{attribute addProperty BoxType "EJ2918-0000-0017"}
{attribute addProperty Id "Module_1_Channel_1_Standard_OutputAT %Q*BOOL811Module_1_Channel_2_Standard_OutputAT %Q*BOOL812Module_1_Channel_3_Standard_OutputAT %Q*BOOL813Module_1_Channel_4_Standard_OutputAT %Q*BOOL814Module_2_Channel_1_Standard_OutputAT %Q*BOOL811Module_2_Channel_2_Standard_OutputAT %Q*BOOL812Module_2_Channel_3_Standard_OutputAT %Q*BOOL813Module_2_Channel_4_Standard_OutputAT %Q*BOOL814"}
{attribute addProperty CRC "3397865097"}
{attribute addProperty SizeInBites "64"}
{attribute addProperty SizeInBytes "8"}
TYPE Outputs_CA874E89 :
STRUCT
	{attribute addProperty Name "Module_1_Channel_1_Standard_Output"}
	Module_1_Channel_1_Standard_Output AT %Q* : BOOL;
	{attribute addProperty Name "Module_1_Channel_2_Standard_Output"}
	Module_1_Channel_2_Standard_Output AT %Q* : BOOL;
	{attribute addProperty Name "Module_1_Channel_3_Standard_Output"}
	Module_1_Channel_3_Standard_Output AT %Q* : BOOL;
	{attribute addProperty Name "Module_1_Channel_4_Standard_Output"}
	Module_1_Channel_4_Standard_Output AT %Q* : BOOL;
	{attribute addProperty Name "Module_2_Channel_1_Standard_Output"}
	Module_2_Channel_1_Standard_Output AT %Q* : BOOL;
	{attribute addProperty Name "Module_2_Channel_2_Standard_Output"}
	Module_2_Channel_2_Standard_Output AT %Q* : BOOL;
	{attribute addProperty Name "Module_2_Channel_3_Standard_Output"}
	Module_2_Channel_3_Standard_Output AT %Q* : BOOL;
	{attribute addProperty Name "Module_2_Channel_4_Standard_Output"}
	Module_2_Channel_4_Standard_Output AT %Q* : BOOL;
END_STRUCT
END_TYPE

(* stored: Version 1.2.0.0, ProductVersion 3.1.4024.9
   DUT Outputs_CA874E89: Id {1fa3f1c5-53cf-4051-923e-476f72a6e698} *)
